// TIA Portal V18 export
// export: Created 2026-06-11T14:52:52.6442991Z, ExportSetting WithDefaults, DisplayName Totally Integrated Automation Portal, DisplayVersion V18, DisplayName TIA Portal Openness, DisplayVersion V18, DisplayName TIA Portal Version Control Interface, DisplayVersion V18, DisplayName STEP 7 Professional, DisplayVersion V18, DisplayName STEP 7 Safety, DisplayVersion V18, DisplayName WinCC Professional, DisplayVersion V18
Screen "Screen_2"  1920x1080, Number=2
  ScreenLayer 
    GraphicView "Graphic view_1" at 0,0 size 1920x1080  Picture=scadabai1_1
    Circle "Circle_1" at 20,151 size 31x31
      RangeAppearanceAnimation "RangeAppearanceAnimation"
        tag 1500S_Trang_Thai
        0..0: back #ffffff, fore #000000
        1..1: back #00ff00, fore #000000
    Circle "Circle_2" at 21,426 size 30x30
      RangeAppearanceAnimation "RangeAppearanceAnimation"
        tag 1404T_Trang_Thai
        0..0: back #ffffff, fore #000000
        1..1: back #00ff00, fore #000000
    Circle "Circle_3" at 130,553 size 31x31
      RangeAppearanceAnimation "RangeAppearanceAnimation"
        tag CR_2013_FO_104_Trang_Thai
        0..0: back #ffffff, fore #000000
        1..1: back #00ff00, fore #000000
    Circle "Circle_4" at 20,751 size 32x32
      RangeAppearanceAnimation "RangeAppearanceAnimation"
        tag BFOC_SS_20_06_Trang_Thai
        0..0: back #ffffff, fore #000000
        1..1: back #00ff00, fore #000000
    IOField "I/O field_1" at 1653,536 size 71x26  DataFormat=Decimal, FormatPattern=99.9, Mode=InOutput
      RangeAppearanceAnimation "RangeAppearanceAnimation"
        tag 1400_TT32_PV
        0..74: back #ffffff, fore #000000
        75..77: back #f59e0b, fore #000000
        78..150: back #dc2626, fore #ffffff, flashing
      ProcessValue := 1400_TT32_PV
    IOField "I/O field_2" at 651,766 size 72x23  DataFormat=Decimal, FormatPattern=99.9, Mode=InOutput
      ProcessValue := 1400_FS51_PV
    IOField "I/O field_3" at 124,828 size 99x20  DataFormat=Decimal, FormatPattern=999.9, Mode=InOutput
      ProcessValue := 1400_LGFE01_PV
    IOField "I/O field_4" at 805,697 size 74x24  DataFormat=Decimal, FormatPattern=99.9, Mode=InOutput
      RangeAppearanceAnimation "RangeAppearanceAnimation"
        tag 1406_TX35_PV
        0..6: back #ffffff, fore #000000
        7..7: back #f59e0b, fore #000000
        8..15: back #dc2626, fore #ffffff, flashing
      ProcessValue := 1406_TX35_PV
    IOField "I/O field_7" at 746,327 size 68x20  DataFormat=Decimal, FormatPattern=999.9, Mode=InOutput
      ProcessValue := 1400_FT101_PV
    IOField "I/O field_8" at 481,270 size 76x24  DataFormat=Decimal, FormatPattern=999.9, Mode=InOutput
      ProcessValue := 1400_FT115_PV
    IOField "I/O field_9" at 1189,265 size 76x26  DataFormat=Decimal, FormatPattern=999.9, Mode=InOutput
      ProcessValue := 1400_1_02_PV
    IOField "I/O field_10" at 1201,887 size 76x25  DataFormat=Decimal, FormatPattern=999.9, Mode=InOutput
      ProcessValue := 1400_FY301_PV
    IOField "I/O field_11" at 1385,537 size 72x23  DataFormat=Decimal, FormatPattern=99.9, Mode=InOutput
      ProcessValue := 1400_TT64_PV
    Circle "Circle_6" at 946,385 size 31x31
      RangeAppearanceAnimation "RangeAppearanceAnimation"
        tag 1400_PT91_Chay
        0..0: back #ffffff, fore #000000
        1..1: back #00ff00, fore #000000
    Circle "Circle_7" at 1756,553 size 31x31
      RangeAppearanceAnimation "RangeAppearanceAnimation"
        tag PC03010T01_Trang_Thai
        0..0: back #ffffff, fore #000000
        1..1: back #00ff00, fore #000000
    Circle "Circle_8" at 1713,676 size 31x31
      RangeAppearanceAnimation "RangeAppearanceAnimation"
        tag 1401_Trang_Thai
        0..0: back #ffffff, fore #000000
        1..1: back #00ff00, fore #000000
    TextField "Text_field_Unit_I/O field_1" at 1732,536 size 50x26  StyleItem=Text field, Text="°C"
    TextField "Text_field_Unit_I/O field_2" at 731,766 size 50x23  StyleItem=Text field, Text="Hz"
    TextField "Text_field_Unit_I/O field_3" at 231,828 size 50x20  StyleItem=Text field, Text="%"
    TextField "Text_field_Unit_I/O field_4" at 887,697 size 20x20  StyleItem=Text field, Text="°C"
    TextField "Text_field_Unit_I/O field_7" at 822,327 size 27x20  StyleItem=Text field, Text="Bar"
    TextField "Text_field_Unit_I/O field_8" at 565,270 size 50x24  StyleItem=Text field, Text="°C"
    TextField "Text_field_Unit_I/O field_9" at 1273,265 size 50x26  StyleItem=Text field, Text="°C"
    TextField "Text_field_Unit_I/O field_10" at 1285,887 size 50x25  StyleItem=Text field, Text="%"
    TextField "Text_field_Unit_I/O field_11" at 1465,537 size 50x23  StyleItem=Text field, Text="°C"
    Rectangle "Header_Bg" at 0,0 size 1920x100  StyleItem=Rectangle
    TextField "Header_Title" at 40,20 size 800x60  StyleItem=Text field, Text="MÀN HÌNH CHÍNH - HỆ THỐNG CÔNG NGHỆ SCADA"
    Button "Header_Alert_TT32" at 840,25 size 110x50  Mode=Text, StyleItem=Button, TextOff="⚠️ TT32 CAO", TextOn="Text"
      RangeAppearanceAnimation "RangeAppearanceAnimation"
        tag 1400_TT32_PV
        0..74: back #0f172a, fore #0f172a
        75..77: back #f59e0b, fore #000000
        78..999: back #dc2626, fore #ffffff, flashing
    Button "Header_Alert_TX35" at 960,25 size 110x50  Mode=Text, StyleItem=Button, TextOff="⚠️ TX35 CAO", TextOn="Text"
      RangeAppearanceAnimation "RangeAppearanceAnimation"
        tag 1406_TX35_PV
        0..6: back #0f172a, fore #0f172a
        7..7: back #f59e0b, fore #000000
        8..999: back #dc2626, fore #ffffff, flashing
    TextField "Header_Operator_Label" at 1100,30 size 250x40  StyleItem=Text field, Text="TÀI KHOẢN VẬN HÀNH:"
    IOField "Header_Operator_Field" at 1360,30 size 160x40  DataFormat=String, FormatPattern=????????????????????, Mode=Output, StyleItem=I/O field
      ProcessValue := @CurrentUser
    Button "Header_Logout_Btn" at 1540,25 size 150x50  Mode=Text, StyleItem=Button, TextOff="ĐĂNG XUẤT", TextOn="Text"
      on Click: Logoff()
    Rectangle "Footer_Bg" at 0,980 size 1920x100  StyleItem=Rectangle
    Button "Footer_Home_Btn" at 200,995 size 400x70  Mode=Text, StyleItem=Button, TextOff="MÀN HÌNH ĐĂNG NHẬP / HOME", TextOn="Text"
      on Click: ActivateScreen(Screen name := Login/out, Object number := 0)
    Button "Footer_SCADA_Btn" at 1320,995 size 400x70  Mode=Text, StyleItem=Button, TextOff="MÀN HÌNH CÔNG NGHỆ (SCADA) - ĐANG XEM", TextOn="Text"
      on Click: ActivateScreen(Screen name := , Object number := 0)
